// TwinCAT 3 PLC project MAS516
// ProgramVersion: 3.1.4023.0
// libraries:
//   Tc2_Standard, * (Beckhoff Automation GmbH)
//   Tc2_System, * (Beckhoff Automation GmbH)
//   Tc3_Module, * (Beckhoff Automation GmbH)
//   VisuDialogs, * (System)
// project tree:
//   DUTs/ E_Status.TcDUT (not stored)
//   Function Blocks/ FB_AnalogInputScaling.TcPOU (not stored), FB_Closedloop.TcPOU, FB_Encoder.TcPOU, FB_JoystickInputScaling.TcPOU (not stored), FB_Openloop.TcPOU, FB_ValveOutput.TcPOU
//   / GlobalTextList.TcGTLO, PlcTask.TcTTO, Visualization Manager.TcVMO (not stored)
//   GVLs/ G_IO.TcGVL, G_Parameters.TcGVL, G_Sensors.TcGVL
//   POUs/ MAIN.TcPOU, P_Inputs.TcPOU, P_Outputs.TcPOU
//   Struct/ ST_AnalogInputScaling.TcDUT (not stored), ST_JoystickInputScaling.TcDUT (not stored), ST_Parameters.TcDUT, ST_ValveDeadBand.TcDUT (not stored), ST_ValveDeadBand_1.TcDUT, ST_ValveOutput.TcDUT (not stored)
//   VISUs/ OpenLoopTest.TcVIS
// real-time tasks:
//   TASK PlcTask: cycle T#10ms, priority 20, ADS port 350
// I/O:
//   DEVICE Device 2 (EtherCAT) (disabled), AmsNetId 192.168.131.1.3.1
//     Term 9 (EK1818) [EK1818 EtherCAT IO-Coupler  (1A E-Bus, 8 Ch. Dig. In, 3ms, 4 Ch. Dig. Out 24V, 0,5A)]
//       Term 10 (EL1008) [EL1008 8Ch. Dig. Input 24V, 3ms]
//       Term 11 (EL3174) [EL3174 4Ch. Ana. Input +/-10V Diff., +/-20mA SingleEnded, 16 Bit]
//       Term 12 (EL3068) [EL3068 8Ch. Ana. Input 0-10V]
//       Term 7 (EL4034) [EL4034 4K. Ana. Ausgang +/-10V, 12bit]
//       Term 14 (EL6751) [EL6751 CANopen Master]
//       Term 17 (EL9011) [EL9011 End Terminal]
//     WinchEncoder (Fraba EtherCAT) [Absolute Rotary Encoder IXARC V01.05]
//     CylinderEncoder (Fraba EtherCAT) [Absolute Rotary Encoder IXARC V01.05]
//   DEVICE Device 1 (EL6751) (disabled), AmsNetId 192.168.131.1.2.1
//     WinchValve (ODC-22)
//     CylinderValve (ODC-22)
// variable links:
//   MAS516/MAS516 Instance <-> Device 2 (EtherCAT)/CylinderEncoder (Fraba EtherCAT)
//     PlcTask Inputs/G_IO.nCylinderEncoderValue <-> Encoder/Position Value
//   MAS516/MAS516 Instance <-> Device 2 (EtherCAT)/Term 9 (EK1818)
//     PlcTask Inputs/G_IO.bEmgOk <-> Channel 1/Input
//     PlcTask Outputs/G_IO.bCylinderValveEnable <-> Channel 12/Output
//     PlcTask Outputs/G_IO.bEnablePCDV <-> Channel 10/Output
//     PlcTask Outputs/G_IO.bOpenBrakes <-> Channel 9/Output
//     PlcTask Outputs/G_IO.bWinchValveEnable <-> Channel 11/Output
//   MAS516/MAS516 Instance <-> Device 2 (EtherCAT)/Term 9 (EK1818)/Term 10 (EL1008)
//     PlcTask Inputs/G_IO.bAutoSwtich <-> Channel 3/Input
//     PlcTask Inputs/G_IO.bCylinderEnable <-> Channel 7/Input
//     PlcTask Inputs/G_IO.bManualSwtich <-> Channel 1/Input
//     PlcTask Inputs/G_IO.bOffSwtich <-> Channel 2/Input
//     PlcTask Inputs/G_IO.bStartButton <-> Channel 4/Input
//     PlcTask Inputs/G_IO.bStopButton <-> Channel 5/Input
//     PlcTask Inputs/G_IO.bWinchEnable <-> Channel 6/Input
//   MAS516/MAS516 Instance <-> Device 2 (EtherCAT)/Term 9 (EK1818)/Term 11 (EL3174)
//     PlcTask Inputs/G_IO.fPDCVMonitor <-> AI Standard Channel 1/Value
//     PlcTask Inputs/G_IO.fPressureWinchA2 <-> AI Standard Channel 2/Value
//     PlcTask Inputs/G_IO.fPressureWinchB <-> AI Standard Channel 3/Value
//     PlcTask Inputs/G_IO.fYoke <-> AI Standard Channel 4/Value
//   MAS516/MAS516 Instance <-> Device 2 (EtherCAT)/Term 9 (EK1818)/Term 12 (EL3068)
//     PlcTask Inputs/G_IO.fJoyXraw <-> AI Standard Channel 6/Value
//     PlcTask Inputs/G_IO.fJoyYraw <-> AI Standard Channel 7/Value
//     PlcTask Inputs/G_IO.fJoyZraw <-> AI Standard Channel 8/Value
//     PlcTask Inputs/G_IO.fPressureCylinderA <-> AI Standard Channel 4/Value
//     PlcTask Inputs/G_IO.fPressureCylinderB <-> AI Standard Channel 5/Value
//     PlcTask Inputs/G_IO.fPressureReturn <-> AI Standard Channel 3/Value
//     PlcTask Inputs/G_IO.fPressureSupply <-> AI Standard Channel 2/Value
//     PlcTask Inputs/G_IO.fPressureWinchA1 <-> AI Standard Channel 1/Value
//   MAS516/MAS516 Instance <-> Device 2 (EtherCAT)/Term 9 (EK1818)/Term 7 (EL4034)
//     PlcTask Outputs/G_IO.fCylValveOut <-> AO Outputs Channel 3/Analog output
//     PlcTask Outputs/G_IO.fWinchPDCVOut <-> AO Outputs Channel 1/Analog output
//     PlcTask Outputs/G_IO.fWinchValveOut <-> AO Outputs Channel 2/Analog output
//   MAS516/MAS516 Instance <-> Device 2 (EtherCAT)/WinchEncoder (Fraba EtherCAT)
//     PlcTask Inputs/G_IO.nWinchEncoderValue <-> Encoder/Position Value

CONFIGURATION MAS516
    RESOURCE PLC ON TwinCAT3
        TASK PlcTask(INTERVAL := T#10ms, PRIORITY := 20);
        PROGRAM MAIN WITH PlcTask : MAIN;
    END_RESOURCE
END_CONFIGURATION

// ---- Struct/ST_Parameters.TcDUT
TYPE ST_Parameters :
STRUCT
	fCyclicTime 					: LREAL := 0.001; // [s]
	fMaxCylVelocityLimit 			: LREAL := 0.005; // [m/s]
	fMaxWinchVelocityLimit 			: LREAL := 0.005; // [rad/s]
	bWinchDeadBandCompOn 			: BOOL := TRUE;
	bCylinderDeadBandCompOn 		: BOOL := TRUE;
	stWinchValveDeadBand 			: ST_ValveDeadBand := (fPosMax := 10000.0, fPosMin := 2000.0, fNegMin := 1500.0, fNegMax := 10000.0);
	stCylValveDeadBand 				: ST_ValveDeadBand := (fPosMax := 10000.0, fPosMin := 2000.0, fNegMin := 2000.0, fNegMax := 7000.0);
	stPressureSensorScaling400bar 	: ST_AnalogInputScaling := (fMaxInputValue := 32767.0, fMinInputValue := 0.0, fMaxOutputValue := 400.0, fMinOutputValue := 0.0);
	stPressureSensorScaling40bar 	: ST_AnalogInputScaling := (fMaxInputValue := 32767.0, fMinInputValue := 0.0, fMaxOutputValue := 40.0, fMinOutputValue := 0.0);
	stJoystickInputScalingX 		: ST_JoystickInputScaling := (fMaxInputValue := 14790.0, fMinInputValue := 1797.0, fNeutralInputValue := 8400, fNeutralDeadband := 50.0, fMaxOutputValue := 1.0, fMinOutputValue := -1.0, fNeutralOutputValue := 0.0);
	stJoystickInputScalingY 		: ST_JoystickInputScaling := (fMaxInputValue := 14770.0, fMinInputValue := 1829.0, fNeutralInputValue := 8340, fNeutralDeadband := 50.0, fMaxOutputValue := 1.0, fMinOutputValue := -1.0, fNeutralOutputValue := 0.0);
	stJoystickInputScalingZ 		: ST_JoystickInputScaling := (fMaxInputValue := 14830.0, fMinInputValue := 1804.0, fNeutralInputValue := 8380, fNeutralDeadband := 50.0, fMaxOutputValue := 1.0, fMinOutputValue := -1.0, fNeutralOutputValue := 0.0);
	stCylPistonPositionScaling 		: ST_AnalogInputScaling := (fMaxInputValue := 32295.0, fMinInputValue := 229.0, fMaxOutputValue := 0.5, fMinOutputValue := 0.0);
	fWinchEncoderOffset 			: LREAL := 0.0; // Encoder value at zero (Cylinder out / second layaer)
	fCylinderEncoderOffset 			: LREAL := 1373.51522; // Encoder value at zero (Cylinder out / second layaer)
	fCylinderDrawWireGearRadius 	: LREAL := 315.23;  // mm/rev
	bEnableWinch 					: BOOL;
	bEnableCylinder					: BOOL;
	V_ref 							: LREAL;  //Velocity Reference
	U   							: LREAL;  //Discharge Area
END_STRUCT
END_TYPE

// ---- Struct/ST_ValveDeadBand_1.TcDUT
TYPE ST_ValveDeadBand_1 :
STRUCT
	fPosMax	: LREAL; // Positive min value [19660..29490]
	fPosMin	: LREAL; // Positive max value [19660..29490]
	fNegMin : LREAL; // Negative max value [9830..19660]
	fNegMax	: LREAL; // Negative min value [9830..19660]
END_STRUCT
END_TYPE

// ---- GVLs/G_IO.TcGVL
{attribute 'qualified_only'}
VAR_GLOBAL
	// Digital Inputs
	bEmgOk 			     AT %I* : BOOL; 
	bStartButton 	     AT %I* : BOOL;
	bStopButton 	     AT %I* : BOOL; 
	bOffSwtich		     AT %I* : BOOL;  
	bManualSwtich	     AT %I* : BOOL; 
	bAutoSwtich			 AT %I* : BOOL; 
	bWinchEnable 		 AT %I* : BOOL; 
	bCylinderEnable 	 AT %I* : BOOL; 
	
	// Analog Intputs
	fJoyXraw 			 AT %I* : INT; 
	fJoyYraw			 AT %I* : INT; 
	fJoyZraw 			 AT %I* : INT; 
	fPDCVMonitor		 AT %I* : INT; 
	fYoke				 AT %I* : INT; 
	fPressureWinchA1 	 AT %I* : INT; 
	fPressureWinchA2 	 AT %I* : INT; 
	fPressureWinchB 	 AT %I* : INT; 
	fPressureCylinderA 	 AT %I* : INT; 
	fPressureCylinderB 	 AT %I* : INT; 
	fPressureSupply 	 AT %I* : INT; 
	fPressureReturn 	 AT %I* : INT; 
	nWinchEncoderValue	 	 AT %I* : UDINT; 
	nCylinderEncoderValue	 AT %I* : UDINT; 
	
	// Digital Outputs
	bOpenBrakes 		 AT %Q* : BOOL; 
	bEnablePCDV 		 AT %Q* : BOOL; 
	bWinchValveEnable 	 AT %Q* : BOOL; 
	bCylinderValveEnable AT %Q* : BOOL; 
	
	// Analog Outputs
	fWinchPDCVOut 		 AT %Q* : INT := 10000; 
	fWinchValveOut 		 AT %Q* : INT; 
	fCylValveOut 		 AT %Q* : INT; 
END_VAR

// ---- GVLs/G_Parameters.TcGVL
{attribute 'qualified_only'}
VAR_GLOBAL
stParam : ST_Parameters;
END_VAR

// ---- GVLs/G_Sensors.TcGVL
{attribute 'qualified_only'}
VAR_GLOBAL
	fJoystickNormalizedY 		: LREAL; 
	fJoystickNormalizedX 		: LREAL; 
	fJoystickNormalizedZ 		: LREAL; 
	fPressureWinchA1 	 		: LREAL; 
	fPressureWinchA2 	 		: LREAL; 
	fPressureWinchB 	 		: LREAL; 
	fPressureCylinderA 	 		: LREAL;  
	fPressureCylinderB 	 		: LREAL; 
	fPressureSupply 	 		: LREAL; 
	fPressureReturn 	 		: LREAL; 
	fWinchEncoderPosition 		: LREAL;
	fCylinderEncoderPosition 	: LREAL;
	fCylinderPosition 			:LREAL;
END_VAR

// ---- POUs/MAIN.TcPOU
PROGRAM MAIN
VAR
	bStatusOk : BOOL;
	bFault : BOOL := FALSE;
	eStatus : E_Status := E_Status.Checking;
	bRunning : BOOL := TRUE;
END_VAR

P_Inputs();
P_Outputs();

IF G_IO.bEmgOk AND NOT(G_IO.bStopButton) AND NOT(G_IO.bOffSwtich) AND NOT(bFault) THEN
	bStatusOk := TRUE;
ELSE 
	bStatusOk := FALSE;
END_IF

CASE eStatus OF 
	E_Status.Checking:
		IF bFault THEN
			eStatus := E_Status.Fault;
		END_IF
		
		IF bStatusOk THEN	
			eStatus := E_Status.Ready;
		END_IF
		
		IF NOT(bStatusOk) THEN	
			eStatus := E_Status.Off;
		END_IF
		
	E_Status.Off:	
		IF bStatusOk THEN	
			eStatus := E_Status.Checking;
		END_IF
		
		IF bFault THEN
			eStatus := E_Status.Fault;
		END_IF

	E_Status.Fault:
		IF NOT(bFault) THEN
			eStatus := E_Status.Checking;
		END_IF
	
	E_Status.Ready:
		IF G_IO.bStartButton AND bStatusOk AND NOT(bFault) THEN
			eStatus := E_Status.Starting;
		END_IF	
		
		IF  NOT(bStatusOk) OR bFault THEN
			eStatus := E_Status.Checking;
		END_IF	

	E_Status.Starting:
		IF bRunning THEN
			eStatus := E_Status.Running;
		END_IF 
		
		IF bFault OR NOT(bStatusOk)  THEN
			eStatus := E_Status.Checking;
		END_IF
		
	
	E_Status.Running:
	
		IF G_IO.bStopButton THEN
			eStatus := E_Status.Stopping;
		END_IF
		
		IF NOT(bRunning) OR NOT(bStatusOk) OR bFault THEN
			eStatus := E_Status.Checking;
		END_IF
	
	E_Status.Stopping:	
		IF NOT(bRunning) THEN
			eStatus := E_Status.Checking;
		END_IF
	
		IF NOT(bStatusOk) OR bFault THEN
		eStatus := E_Status.Checking;
		END_IF	
	
ELSE 	
	eStatus := E_Status.Checking;
END_CASE

END_PROGRAM

// ---- POUs/P_Inputs.TcPOU
PROGRAM P_Inputs
VAR
	fbJoystickWinch 				: FB_JoystickInputScaling;
	fbJoystickCyl 					: FB_JoystickInputScaling;
	fbJoystickRot 					: FB_JoystickInputScaling;
	fbWinchPosition 				: FB_Encoder;
	fbCylinderPosition 				: FB_Encoder;
	fbCylPistonPosition 			: FB_AnalogInputScaling;
	fbPressureSupply 				: FB_AnalogInputScaling;
	fbPressureReturn 				: FB_AnalogInputScaling;
	fbPressureCyl_A_PistonSide 		: FB_AnalogInputScaling;
	fbPressureCyl_B_RodSide			: FB_AnalogInputScaling;
	fbPressureWinch_A1_Input 		: FB_AnalogInputScaling;
	fbPressureWinch_A2_Input 		: FB_AnalogInputScaling;
	fbPressureWinch_B_Output		: FB_AnalogInputScaling;
	eStatus : E_Status;
END_VAR

fbJoystickWinch(
	bEnable := G_IO.bManualSwtich,
	nRawInput := G_IO.fJoyYraw,
	stJoystickInputScaling := G_Parameters.stParam.stJoystickInputScalingY,
	fNormalizedOutput => G_Sensors.fJoystickNormalizedY
);

fbJoystickCyl(
	bEnable := G_IO.bManualSwtich,
	nRawInput := G_IO.fJoyXraw,
	stJoystickInputScaling := G_Parameters.stParam.stJoystickInputScalingX,
	fNormalizedOutput => G_Sensors.fJoystickNormalizedX
);

fbJoystickRot(
	bEnable := G_IO.bManualSwtich,
	nRawInput := G_IO.fJoyZraw,
	stJoystickInputScaling := G_Parameters.stParam.stJoystickInputScalingZ,
	fNormalizedOutput => G_Sensors.fJoystickNormalizedZ
);

fbWinchPosition (
	nRawInput := G_IO.nWinchEncoderValue, 
	fEncoderOffset := G_Parameters.stParam.fWinchEncoderOffset,
	fPosition => G_Sensors.fWinchEncoderPosition
);

fbCylinderPosition (
	nRawInput := G_IO.nCylinderEncoderValue, 
	fEncoderOffset := G_Parameters.stParam.fCylinderEncoderOffset,
	fPosition => G_Sensors.fCylinderEncoderPosition
);

//G_Sensors.fWinchWirePosition := fbWinchPosition.fPosition*G_Parameters.stParam.fWinchDrumScaling;
G_Sensors.fCylinderPosition := -(fbCylinderPosition.fPosition/360)*G_Parameters.stParam.fCylinderDrawWireGearRadius*0.001;


fbPressureSupply(
	nRawInput := G_IO.fPressureSupply,
	stAnalogInputScaling := G_Parameters.stParam.stPressureSensorScaling400bar,
	fOutput => G_Sensors.fPressureSupply
);

fbPressureReturn(
	nRawInput := G_IO.fPressureReturn,
	stAnalogInputScaling := G_Parameters.stParam.stPressureSensorScaling40bar,
	fOutput => G_Sensors.fPressureReturn
);

fbPressureCyl_A_PistonSide(
	nRawInput := G_IO.fPressureCylinderA,
	stAnalogInputScaling := G_Parameters.stParam.stPressureSensorScaling400bar,
	fOutput => G_Sensors.fPressureCylinderA
);

fbPressureCyl_B_RodSide(
	nRawInput := G_IO.fPressureCylinderB,
	stAnalogInputScaling := G_Parameters.stParam.stPressureSensorScaling400bar,
	fOutput => G_Sensors.fPressureCylinderB
);

fbPressureWinch_A1_Input(
	nRawInput := G_IO.fPressureWinchA1,
	stAnalogInputScaling := G_Parameters.stParam.stPressureSensorScaling400bar,
	fOutput => G_Sensors.fPressureWinchA1
);

fbPressureWinch_A2_Input(
	nRawInput := G_IO.fPressureWinchA2,
	stAnalogInputScaling := G_Parameters.stParam.stPressureSensorScaling400bar,
	fOutput => G_Sensors.fPressureWinchA2
);

fbPressureWinch_B_Output(
	nRawInput := G_IO.fPressureWinchB,
	stAnalogInputScaling := G_Parameters.stParam.stPressureSensorScaling400bar,
	fOutput => G_Sensors.fPressureWinchB
);

END_PROGRAM

// ---- Function Blocks/FB_Encoder.TcPOU
FUNCTION_BLOCK FB_Encoder
VAR_INPUT
	nRawInput : UDINT;
	fEncoderOffset : LREAL; 
END_VAR
VAR_OUTPUT
	fPosition 		: LREAL;
END_VAR
VAR PERSISTENT
	nRounds			: DINT;
	nRawLast 		: DINT;
END_VAR	
VAR
	nInput 		: DINT;
	nTempInputDiff	: DINT;
	nCount 			: DINT;
	nMaxValue30bit 	: DINT :=  1073741823; // 2^30 - 1	
	nThreshold30bit	: DINT := nMaxValue30bit/2;
	fScale16bit		: LREAL := 360.0/65535.0; // 360deg/(2^16 - 1)
	fTempPosition   : LREAL;
END_VAR

// Convert to DINT (same as const values)
nInput := UDINT_TO_DINT(nRawInput);

// Define Encoder Rounds
nTempInputDiff := nInput - nRawLast;
IF (nTempInputDiff > nThreshold30bit) THEN
	nRounds := nRounds - 1;
END_IF

IF (nTempInputDiff < -nThreshold30bit) THEN
	nRounds := nRounds + 1;
END_IF

// Count Encoder Rounds
nCount := nInput + nRounds*nMaxValue30bit;

//Position Output
fPosition := DINT_TO_LREAL(nCount)*fScale16bit - fEncoderOffset; // [deg]

END_FUNCTION_BLOCK

// ---- POUs/P_Outputs.TcPOU
PROGRAM P_Outputs
VAR
	fbWinchValveOutput 		: FB_ValveOutput;
	fbCylValveOutput 		: FB_ValveOutput;
	fbOpenloop				: FB_Openloop;
	eStatus 				: E_Status; 
	bEnableWinch 			: BOOL;
	bTest1 : BOOL;
	bTest2 : BOOL;
	ValveOpening 			: LREAL;
END_VAR

IF MAIN.eStatus = E_Status.Running THEN
	G_IO.bEnablePCDV := TRUE;
	G_IO.bWinchValveEnable := TRUE;
	G_IO.bCylinderValveEnable := TRUE;
ELSE
	G_IO.bEnablePCDV := FALSE;	
	G_IO.bWinchValveEnable := FALSE;
	G_IO.bCylinderValveEnable := FALSE;
END_IF

///////////////////// Winch //////////////////////////////
IF (MAIN.eStatus = E_Status.Running) AND G_IO.bWinchEnable THEN 
	G_IO.bOpenBrakes := TRUE;
	bEnableWinch := TRUE;
ELSE
	G_IO.bOpenBrakes := FALSE;
	bEnableWinch := FALSE;
END_IF

fbWinchValveOutput(
	bEnable := bEnableWinch,
	bDeadBandCompOn := G_Parameters.stParam.bWinchDeadBandCompOn,
	stValveDeadBand := G_Parameters.stParam.stWinchValveDeadBand,
	fNormalizedInput := G_Sensors.fJoystickNormalizedY,
	nOutput => G_IO.fWinchValveOut
);

///////////////////// Cylinder //////////////////////////////

IF (MAIN.eStatus = E_Status.Running) AND G_IO.bCylinderEnable THEN 
	G_Parameters.stParam.bEnableCylinder := TRUE;
ELSE
	G_Parameters.stParam.bEnableCylinder := FALSE;
END_IF

fbCylValveOutput(
	bEnable := G_Parameters.stParam.bEnableCylinder,
	bDeadBandCompOn := G_Parameters.stParam.bCylinderDeadBandCompOn,
	stValveDeadBand := G_Parameters.stParam.stCylValveDeadBand,
	fNormalizedInput := G_Sensors.fJoystickNormalizedX,
	nOutput => G_IO.fCylValveOut
);

fbOpenloop(
	U => G_Parameters.stParam.U
);

END_PROGRAM

// ---- Function Blocks/FB_ValveOutput.TcPOU
FUNCTION_BLOCK FB_ValveOutput
VAR_INPUT
	bEnable 			: BOOL;
	bDeadBandCompOn 	: BOOL;
	stValveDeadBand 	: ST_ValveDeadBand;
	fNormalizedInput 	: LREAL;
END_VAR
VAR_OUTPUT
	bEnableValveOutput : BOOL;
	nOutput : INT; 
END_VAR
VAR
	nOffset 	: INT := 0;
	nMaxValue	: INT := 32767;
	nMinValue 	: INT :=  -32767;
	nTempOutput : INT;
END_VAR

IF	bDeadBandCompOn THEN
	IF fNormalizedInput > 0.0 THEN
		nTempOutput := LREAL_TO_INT(fNormalizedInput*(stValveDeadBand.fPosMax - stValveDeadBand.fPosMin) + stValveDeadBand.fPosMin);
	ELSIF fNormalizedInput < 0.0 THEN
		nTempOutput := LREAL_TO_INT(fNormalizedInput*(stValveDeadBand.fNegMax - stValveDeadBand.fNegMin) - stValveDeadBand.fNegMin);
	ELSE
		nTempOutput := 0;
	END_IF
ELSE
	IF fNormalizedInput > 0.0 THEN
		nTempOutput := LREAL_TO_INT(fNormalizedInput*32767.0);
	ELSIF fNormalizedInput < 0.0 THEN
		nTempOutput := LREAL_TO_INT(fNormalizedInput *32767.0);
	ELSE
		nTempOutput := 0;
	END_IF	
END_IF	

IF bEnable THEN
	nOutput := LIMIT(nMinValue, nTempOutput, nMaxValue);
	bEnableValveOutput := TRUE; 
ELSE 	
	nOutput := 0;
	bEnableValveOutput := FALSE;	
END_IF

END_FUNCTION_BLOCK

// ---- Function Blocks/FB_Openloop.TcPOU
FUNCTION_BLOCK FB_Openloop
VAR_INPUT
END_VAR
VAR_OUTPUT
	U : LREAL;  //Discharge Area - Valve
	ValveOutput : LREAL; 
END_VAR
VAR
	BoreArea : LREAL := 0.0031172426775;
	AnnulusArea : LREAL := 0.0018606066775;
	MaxFlow : LREAL := 25;
END_VAR

IF ((* G_Parameters.stParam.bEnableCylinder := TRUE AND *) G_Parameters.stParam.V_ref > 0) THEN
	U := (60000 * G_Parameters.stParam.V_ref * BoreArea) / MaxFlow;
	
ELSIF ((*G_Parameters.stParam.bEnableCylinder := TRUE AND *)G_Parameters.stParam.V_ref < 0) THEN
	U := (60000 * G_Parameters.stParam.V_ref * AnnulusArea) / MaxFlow;
	
ELSE 
	U := 0;
END_IF

END_FUNCTION_BLOCK

// ---- Function Blocks/FB_Closedloop.TcPOU
FUNCTION_BLOCK FB_Closedloop
VAR_INPUT
END_VAR
VAR_OUTPUT
END_VAR
VAR
END_VAR

END_FUNCTION_BLOCK

// ---- GlobalTextList.TcGTLO
TEXTLIST GlobalTextList
  396 = '%f'
  594 = '%i'
  706 = '%s'
  721 = 'Dishcarge Area'
  771 = 'Input Velocity'
  752 = 'U'
  161 = 'Velocity Reference'
END_TEXTLIST

// ---- VISUs/OpenLoopTest.TcVIS
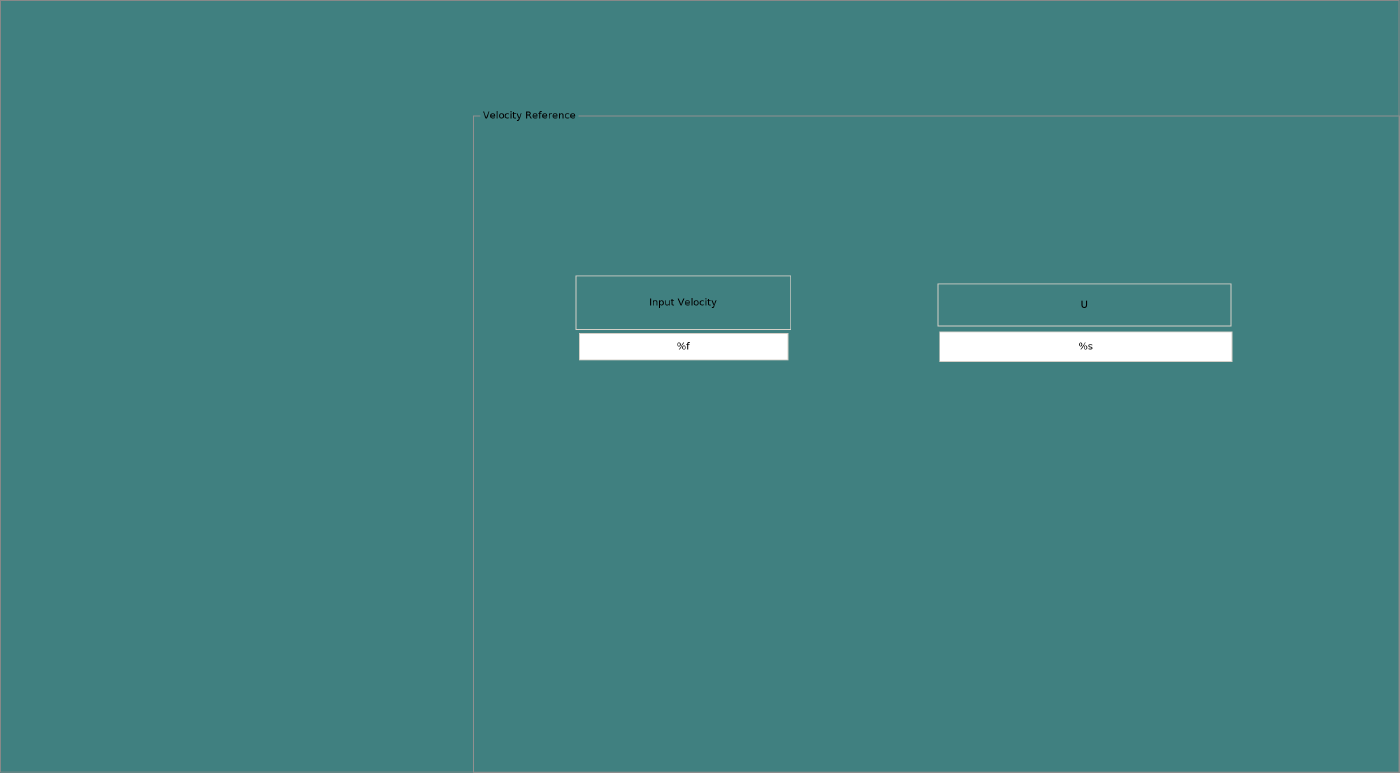
VISUALIZATION OpenLoopTest  // 1574x870
    GroupBox (532,122 1042x748), "Velocity Reference"
        Textfield (119,253 235x30), "%f", text variable: G_Parameters.stParam.V_ref
            OnMouseClick: write the text variable via Default
        Textfield (524,251 329x34), "%s", text variable: G_Parameters.stParam.U
        Textfield (115,188 242x61), "Input Velocity"
        Textfield (522,197 330x48), "U"
END_VISUALIZATION
